// TIA Portal V20 export
// export: Created 2026-04-11T06:02:30.080907Z, ExportSetting WithDefaults, DisplayName Totally Integrated Automation Portal, DisplayVersion V20, DisplayName TIA Portal Openness, DisplayVersion V20, DisplayName TIA Portal Version Control Interface, DisplayVersion V20, DisplayName STEP 7 Professional, DisplayVersion V20, DisplayName STEP 7 Safety, DisplayVersion V20, DisplayName WinCC Basic/Comfort/Advanced, DisplayVersion V20, DisplayName WinCC Unified, DisplayVersion V20
TYPE "udtError_Hopper"
// stored: IsFailsafeCompliant false
   STRUCT
      LowLevelSignalFailure { ExternalWritable := 'False'} : Bool;   // High level sensor is ON, but Low level sensor still OFF.
      LowPressureSignalFailure { ExternalWritable := 'False'} : Bool;   // High pressure sensor is ON, but Low pressure sensor still OFF.
      HighPressure { ExternalWritable := 'False'} : Bool;   // Differential pressure High timeout. Filters may be plugged.
      LowPressure { ExternalWritable := 'False'} : Bool;   // Differential pressure Low timeout. Inspect filters for holes.
      HighLevel { ExternalWritable := 'False'} : Bool;   // Hopper High Level Alarm
      LowLevel { ExternalWritable := 'False'} : Bool;   // Hopper Low Level Alarm
   END_STRUCT;
END_TYPE
